(* Logix 5000 project; controller p65 vendor 1 type 14 code 85 rev 20.11; software revision 20.01; part 2 of 7 *)
(* tags used below, declared in another part *)
   BatterybattCurrent : ALIAS FOR REAL00_0;
   BatterybattCurrentHILS : ALIAS FOR plc1_local_3[4];
   Batterybattcurrentoffset : REAL;
   BatterybattCurrentRaw : ALIAS FOR Local:1:I.Ch4Data;
   BatterybattPower : ALIAS FOR REAL00_1;
   BatterybattVoltage : ALIAS FOR REAL00_2;
   BatterybattVoltageHILS : ALIAS FOR plc1_local_3[5];
   BatterybattVoltageRaw : ALIAS FOR Local:1:I.Ch0Data;
   BatterycanSupplyPower : ALIAS FOR DINT00_22.0;
   Batterycharge : ALIAS FOR REAL00_3;
   BatterychargeCurrent : ALIAS FOR REAL00_4;
   BatterychargeToGo : ALIAS FOR REAL00_5;
   BatterychargingTimer : ALIAS FOR CLTIMER00_0;
   BatterycomputeAddition : ALIAS FOR DINT00_22.7;
   BatterycomputeSubtraction : ALIAS FOR DINT00_22.8;
   BatterydecideToCharge : ALIAS FOR DINT00_22.15;
   BatterydecideToDisconnect : ALIAS FOR DINT00_22.16;
   BatterydeltaCharge : ALIAS FOR REAL00_6;
   BatterydischargeCurrent : ALIAS FOR REAL00_7;
   BatterydischargingTimer : ALIAS FOR CLTIMER00_1;
   BatterydisconnectedTimer : ALIAS FOR CLTIMER00_2;
   Batteryefficiency : ALIAS FOR REAL00_8;
   Batteryfraction : ALIAS FOR REAL00_9;
   BatteryfractionCharged : ALIAS FOR REAL00_10;
   BatteryfractionChargedEstimate : ALIAS FOR REAL00_11;
   BatteryfractionToGo : ALIAS FOR REAL00_12;
   BatteryfullCharge : ALIAS FOR REAL00_13;
   BatteryfullChargeCurrent : ALIAS FOR REAL00_14;
   BatterygeneralTimer : ALIAS FOR CLTIMER00_3;
   BatterygridCurrent : ALIAS FOR REAL00_15;
   BatterygridCurrentabs : REAL;
   BatterygridCurrentHILS : ALIAS FOR plc1_local_3[2];
   Batterygridcurrentoffset : REAL;
   BatterygridCurrentRaw : ALIAS FOR Local:1:I.Ch5Data;
   BatterygridPower : ALIAS FOR REAL00_16;
   BatterygridVoltage : ALIAS FOR REAL00_17;
   BatterygridVoltageHILS : ALIAS FOR plc1_local_3[3];
   BatterygridVoltageRaw : ALIAS FOR Local:1:I.Ch9Data;
   BatteryintReqCharge : ALIAS FOR DINT00_22.17;
   BatteryintReqDischarge : ALIAS FOR DINT00_22.18;
   BatteryintReqDisconnect : ALIAS FOR DINT00_22.19;
   BatteryisCharging : ALIAS FOR DINT00_22.20;
   BatteryisDischarging : ALIAS FOR DINT00_22.21;
   BatteryisDisconnected : ALIAS FOR DINT00_22.22;
   BatteryisFullyCharged : ALIAS FOR DINT00_22.23;
   BatteryisFunctional : ALIAS FOR DINT00_22.24;
   BatterylastChargingTime : ALIAS FOR DINT00_0;
   BatterylastDischargingTime : ALIAS FOR DINT00_1;
   BatterylastDisconnectedTime : ALIAS FOR DINT00_2;
   BatterylastFractionChargedDelta : ALIAS FOR REAL00_18;
   BatterylastIntReqCharge : ALIAS FOR DINT00_22.25;
   BatterylastIntReqDischarge : ALIAS FOR DINT00_22.26;
   BatterylastIntReqDisconnect : ALIAS FOR DINT00_22.27;
   BatterylowestSOC : ALIAS FOR REAL00_19;
   Batterymultiplier : ALIAS FOR REAL00_20;
   BatterynominalDischargeCurrent : ALIAS FOR REAL00_21;
   BatteryocVoltage : ALIAS FOR REAL00_22;
   BatteryoutOfOperationalRange : ALIAS FOR DINT00_22.28;
   BatterypeukertLessOne : ALIAS FOR REAL00_23;
   Batteryproduct : ALIAS FOR REAL00_24;
   BatteryreqCharge : ALIAS FOR DINT00_22.29;
   BatteryreqDischarge : ALIAS FOR DINT00_22.30;
   BatteryreqDisconnect : ALIAS FOR DINT00_22.31;
   BatteryreqInitialize : ALIAS FOR DINT00_23.0;
   BatterysettlingTimer : ALIAS FOR CLTIMER00_4;
   Batterysoc : ALIAS FOR REAL00_25;
   BatterysocToGo : ALIAS FOR REAL00_26;
   BatterySOCTooLowEventFail : ALIAS FOR DINT00_23.1;
   BatterySOCTooLowEventSuccess : ALIAS FOR DINT00_23.2;
   BatterySOCTooLowFailTimer : ALIAS FOR CLTIMER00_5;
   BatterySOCTooLowInProcess : ALIAS FOR DINT00_23.3;
   BatterySOCTooLowMsg : ALIAS FOR MESSAGE00_0;
   BatterySOCTooLowSuccessTimer : ALIAS FOR CLTIMER00_6;
   BatterytimeSinceLastMeasurement : ALIAS FOR REAL00_27;
   BatterytimeToLowestSOC : ALIAS FOR REAL00_28;
   BatteryunambiguousCommand : ALIAS FOR DINT00_23.4;
   CBclose : ALIAS FOR Local:3:O.Data.15;
   CBcloseHILS : ALIAS FOR plc1_local_6[0].14;
   CBcloseProxy : ALIAS FOR DINT00_22.1;
   CBintReqClose : ALIAS FOR DINT00_22.2;
   CBisClosed : ALIAS FOR DINT00_22.3;
   CBisOpen : ALIAS FOR DINT00_22.4;
   CBreqClose : ALIAS FOR DINT00_22.5;
   CBreqOpen : ALIAS FOR DINT00_22.6;
   Commaccum : ALIAS FOR REAL00_31;
   CommBattempt : ALIAS FOR DINT00_3;
   CommBclose : ALIAS FOR Local:3:O.Data.11;
   CommBcloseHILS : ALIAS FOR plc1_local_6[0].11;
   CommBcloseProxy : ALIAS FOR DINT00_23.12;
   CommBdeadBand : ALIAS FOR REAL00_32;
   CommBfailedToOpen : ALIAS FOR DINT00_23.13;
   CommBintForceOpen : ALIAS FOR DINT00_23.14;
   CommBintReqClose : ALIAS FOR DINT00_23.15;
   CommBisClosed : ALIAS FOR DINT00_23.16;
   CommBisOpen : ALIAS FOR DINT00_23.17;
   CommBmaxAttempts : ALIAS FOR DINT00_4;
   CommBmaxLoadCurrent : ALIAS FOR REAL00_33;
   CommBopenTimer : ALIAS FOR CLTIMER00_7;
   CommBreqClose : ALIAS FOR DINT00_23.18;
   CommBreqOpen : ALIAS FOR DINT00_23.19;
   CommBreqReset : ALIAS FOR DINT00_23.20;
   CommBretriesFailed : ALIAS FOR DINT00_23.21;
   CommBtooMuchCurrent : ALIAS FOR DINT00_23.22;
   CommBunexpectedLowCurrent : ALIAS FOR DINT00_23.23;
   CommcanNotifyUser : ALIAS FOR DINT00_23.24;
   CommcommandChanged : ALIAS FOR DINT00_23.25;
   CommcommandChangedTimer : ALIAS FOR CLTIMER00_8;
   Commcurrent : ALIAS FOR REAL00_34;
   CommcurrentHILS : ALIAS FOR plc1_local_3[8];
   CommcurrentRaw : ALIAS FOR Local:1:I.Ch10Data;
   Commdeadband : ALIAS FOR REAL00_35;
   Commdifference : ALIAS FOR REAL00_36;
   CommfailedToConnect : ALIAS FOR DINT00_23.26;
   CommfailedToDisconnect : ALIAS FOR DINT00_23.27;
   CommintReqConnect : ALIAS FOR DINT00_23.28;
   CommisConnected : ALIAS FOR DINT00_23.29;
   CommisDisconnected : ALIAS FOR DINT00_23.30;
   CommnotificationTimer : ALIAS FOR CLTIMER00_44;
   CommOverCurrentConditionEventFail : ALIAS FOR DINT00_27.13;
   CommOverCurrentConditionEventSuccess : ALIAS FOR DINT00_27.14;
   CommOverCurrentConditionFailTimer : ALIAS FOR CLTIMER00_45;
   CommOverCurrentConditionInProcess : ALIAS FOR DINT00_27.15;
   CommOverCurrentConditionMsg : ALIAS FOR MESSAGE00_11;
   CommOverCurrentConditionSuccessTimer : ALIAS FOR CLTIMER00_46;
   Commpower : ALIAS FOR REAL00_102;
   CommreqConnect : ALIAS FOR DINT00_27.16;
   CommreqDisconnect : ALIAS FOR DINT00_27.17;
   CommsampleNow : ALIAS FOR DINT00_27.18;
   CommsampleTimer : ALIAS FOR CLTIMER00_47;
   Commtotal : ALIAS FOR REAL00_103;
   CommtotalTooLarge : ALIAS FOR DINT00_27.19;
   CommtotalTooSmall : ALIAS FOR DINT00_27.20;
   CommuserNotified : ALIAS FOR DINT00_27.21;
   Commvoltage : ALIAS FOR REAL00_104;
   CommvoltageHILS : ALIAS FOR plc1_local_3[9];
   CommvoltageRaw : ALIAS FOR Local:2:I.Ch7Data;
   DBclose : ALIAS FOR Local:3:O.Data.14;
   DBcloseHILS : ALIAS FOR plc1_local_6[0].13;
   DBcloseProxy : ALIAS FOR DINT00_22.9;
   DBintReqClose : ALIAS FOR DINT00_22.10;
   DBisClosed : ALIAS FOR DINT00_22.11;
   DBisOpen : ALIAS FOR DINT00_22.12;
   DBreqClose : ALIAS FOR DINT00_22.13;
   DBreqOpen : ALIAS FOR DINT00_22.14;
   DCMicroGridisSimulating : ALIAS FOR DINT00_23.10;
   DCMicroGridsourcesProvidingExcessPower : ALIAS FOR DINT00_33.7;
   Load01current : ALIAS FOR REAL00_39;
   Load02current : ALIAS FOR REAL00_52;
   Load03current : ALIAS FOR REAL00_65;
   Load04current : ALIAS FOR REAL00_78;
   Load05current : ALIAS FOR REAL00_91;
   LoadslowVoltage : ALIAS FOR DINT00_27.23;
   UsingAgents : BOOL;

PROGRAM Battery   (* main routine Battery *)

ROUTINE Battery   (* ladder *)
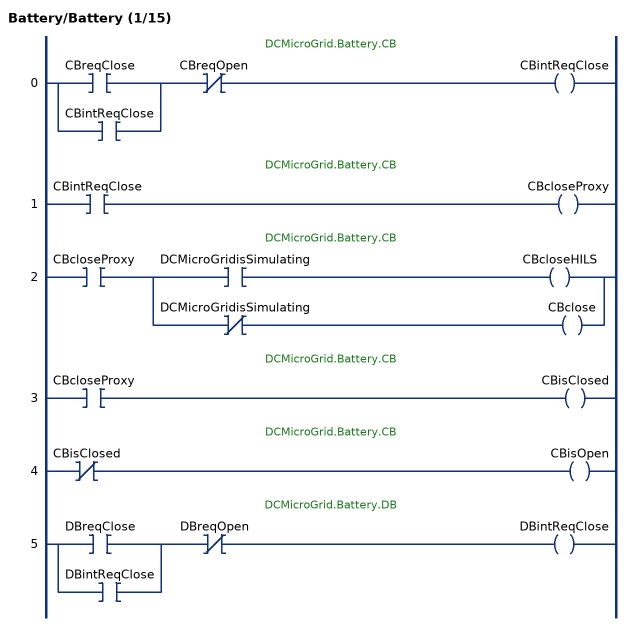
   // DCMicroGrid.Battery.CB
   0: [XIC(CBreqClose) ,XIC(CBintReqClose) ]XIO(CBreqOpen)OTE(CBintReqClose);
   // DCMicroGrid.Battery.CB
   1: XIC(CBintReqClose)OTE(CBcloseProxy);
   // DCMicroGrid.Battery.CB
   2: XIC(CBcloseProxy)[XIC(DCMicroGridisSimulating) OTE(CBcloseHILS) ,XIO(DCMicroGridisSimulating) OTE(CBclose) ];
   // DCMicroGrid.Battery.CB
   3: XIC(CBcloseProxy)OTE(CBisClosed);
   // DCMicroGrid.Battery.CB
   4: XIO(CBisClosed)OTE(CBisOpen);
   // DCMicroGrid.Battery.DB
   5: [XIC(DBreqClose) ,XIC(DBintReqClose) ]XIO(DBreqOpen)OTE(DBintReqClose);
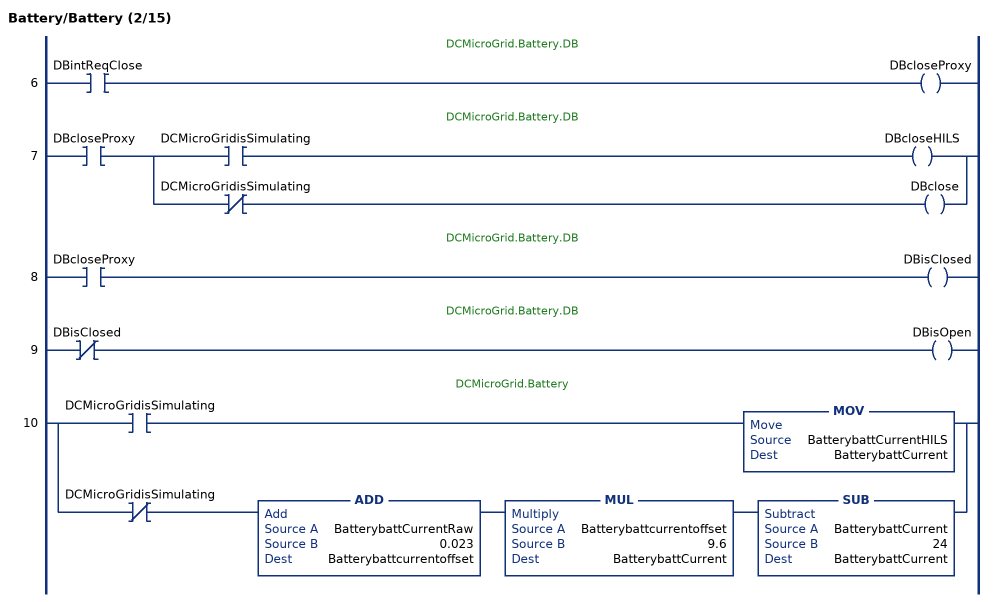
   // DCMicroGrid.Battery.DB
   6: XIC(DBintReqClose)OTE(DBcloseProxy);
   // DCMicroGrid.Battery.DB
   7: XIC(DBcloseProxy)[XIC(DCMicroGridisSimulating) OTE(DBcloseHILS) ,XIO(DCMicroGridisSimulating) OTE(DBclose) ];
   // DCMicroGrid.Battery.DB
   8: XIC(DBcloseProxy)OTE(DBisClosed);
   // DCMicroGrid.Battery.DB
   9: XIO(DBisClosed)OTE(DBisOpen);
   // DCMicroGrid.Battery
   10: [XIC(DCMicroGridisSimulating) MOV(BatterybattCurrentHILS,BatterybattCurrent) ,XIO(DCMicroGridisSimulating) ADD(BatterybattCurrentRaw,0.023,Batterybattcurrentoffset) MUL(Batterybattcurrentoffset,9.6,BatterybattCurrent) SUB(BatterybattCurrent,24,BatterybattCurrent) ];
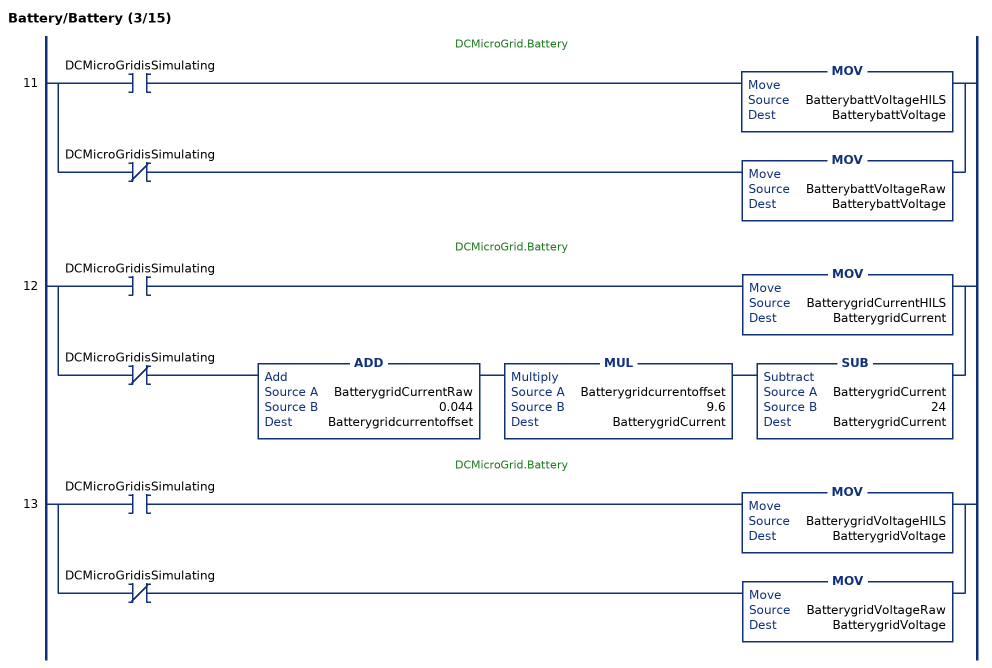
   // DCMicroGrid.Battery
   11: [XIC(DCMicroGridisSimulating) MOV(BatterybattVoltageHILS,BatterybattVoltage) ,XIO(DCMicroGridisSimulating) MOV(BatterybattVoltageRaw,BatterybattVoltage) ];
   // DCMicroGrid.Battery
   12: [XIC(DCMicroGridisSimulating) MOV(BatterygridCurrentHILS,BatterygridCurrent) ,XIO(DCMicroGridisSimulating) ADD(BatterygridCurrentRaw,0.044,Batterygridcurrentoffset) MUL(Batterygridcurrentoffset,9.6,BatterygridCurrent) SUB(BatterygridCurrent,24,BatterygridCurrent) ];
   // DCMicroGrid.Battery
   13: [XIC(DCMicroGridisSimulating) MOV(BatterygridVoltageHILS,BatterygridVoltage) ,XIO(DCMicroGridisSimulating) MOV(BatterygridVoltageRaw,BatterygridVoltage) ];
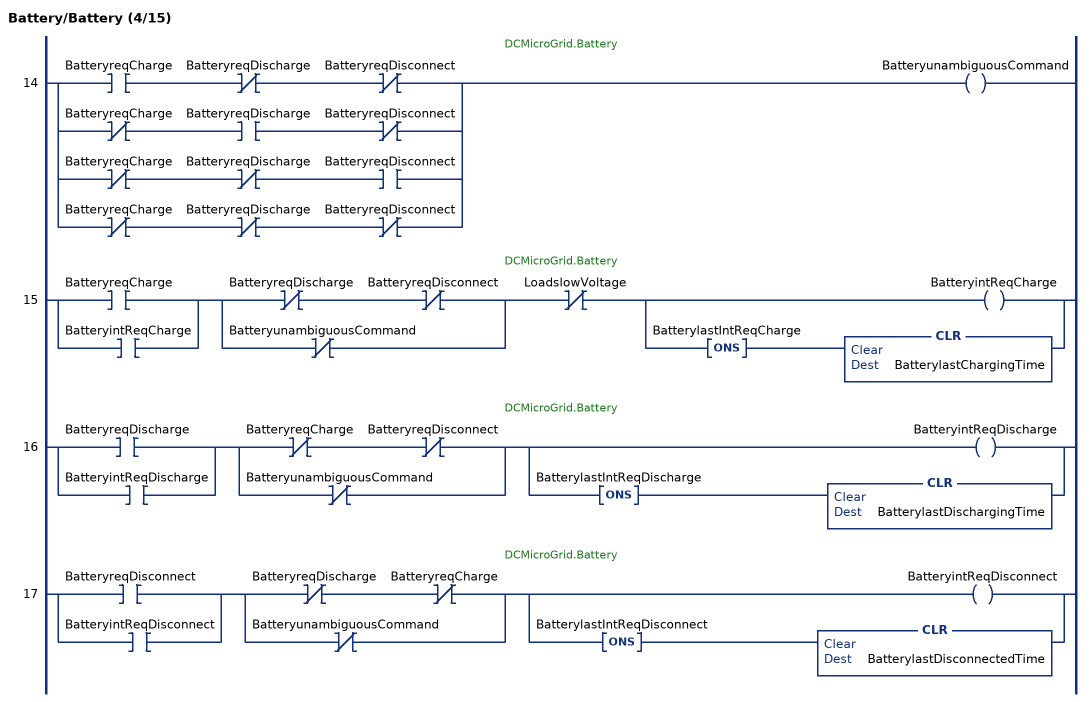
   // DCMicroGrid.Battery
   14: [XIC(BatteryreqCharge) XIO(BatteryreqDischarge) XIO(BatteryreqDisconnect) ,XIO(BatteryreqCharge) XIC(BatteryreqDischarge) XIO(BatteryreqDisconnect) ,XIO(BatteryreqCharge) XIO(BatteryreqDischarge) XIC(BatteryreqDisconnect) ,XIO(BatteryreqCharge) XIO(BatteryreqDischarge) XIO(BatteryreqDisconnect) ]OTE(BatteryunambiguousCommand);
   // DCMicroGrid.Battery
   15: [XIC(BatteryreqCharge) ,XIC(BatteryintReqCharge) ][XIO(BatteryreqDischarge) XIO(BatteryreqDisconnect) ,XIO(BatteryunambiguousCommand) ]XIO(LoadslowVoltage)[OTE(BatteryintReqCharge) ,ONS(BatterylastIntReqCharge) CLR(BatterylastChargingTime) ];
   // DCMicroGrid.Battery
   16: [XIC(BatteryreqDischarge) ,XIC(BatteryintReqDischarge) ][XIO(BatteryreqCharge) XIO(BatteryreqDisconnect) ,XIO(BatteryunambiguousCommand) ][OTE(BatteryintReqDischarge) ,ONS(BatterylastIntReqDischarge) CLR(BatterylastDischargingTime) ];
   // DCMicroGrid.Battery
   17: [XIC(BatteryreqDisconnect) ,XIC(BatteryintReqDisconnect) ][XIO(BatteryreqDischarge) XIO(BatteryreqCharge) ,XIO(BatteryunambiguousCommand) ][OTE(BatteryintReqDisconnect) ,ONS(BatterylastIntReqDisconnect) CLR(BatterylastDisconnectedTime) ];
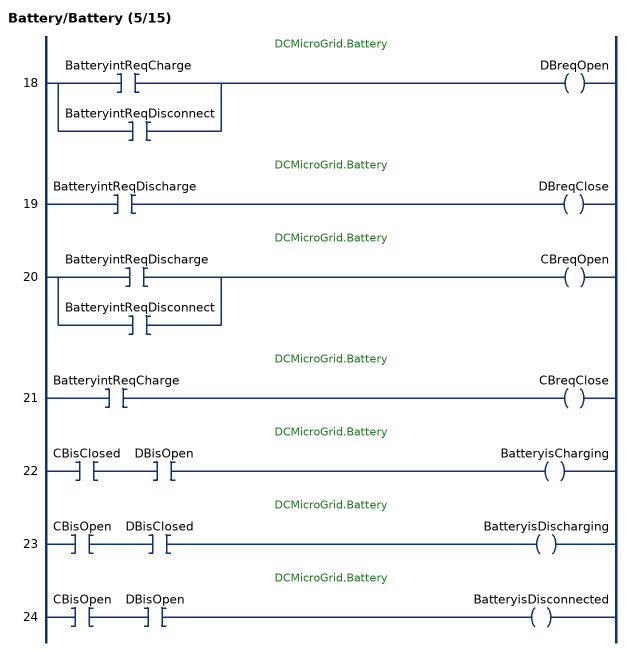
   // DCMicroGrid.Battery
   18: [XIC(BatteryintReqCharge) ,XIC(BatteryintReqDisconnect) ]OTE(DBreqOpen);
   // DCMicroGrid.Battery
   19: XIC(BatteryintReqDischarge)OTE(DBreqClose);
   // DCMicroGrid.Battery
   20: [XIC(BatteryintReqDischarge) ,XIC(BatteryintReqDisconnect) ]OTE(CBreqOpen);
   // DCMicroGrid.Battery
   21: XIC(BatteryintReqCharge)OTE(CBreqClose);
   // DCMicroGrid.Battery
   22: XIC(CBisClosed)XIC(DBisOpen)OTE(BatteryisCharging);
   // DCMicroGrid.Battery
   23: XIC(CBisOpen)XIC(DBisClosed)OTE(BatteryisDischarging);
   // DCMicroGrid.Battery
   24: XIC(CBisOpen)XIC(DBisOpen)OTE(BatteryisDisconnected);
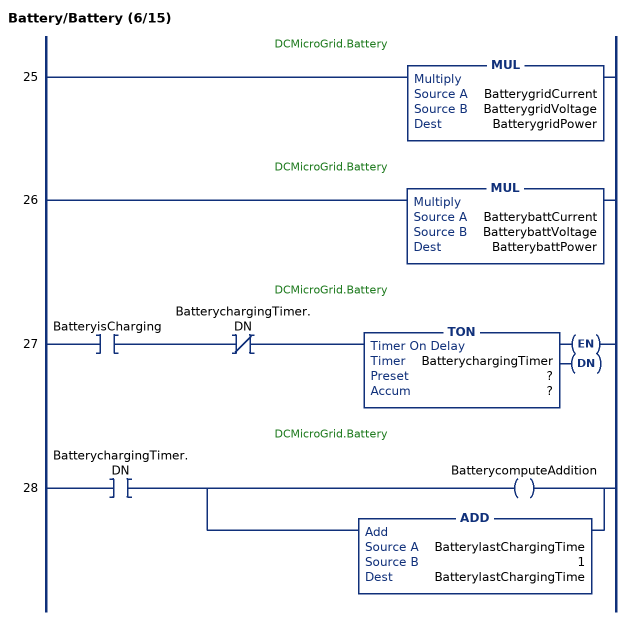
   // DCMicroGrid.Battery
   25: MUL(BatterygridCurrent,BatterygridVoltage,BatterygridPower);
   // DCMicroGrid.Battery
   26: MUL(BatterybattCurrent,BatterybattVoltage,BatterybattPower);
   // DCMicroGrid.Battery
   27: XIC(BatteryisCharging)XIO(BatterychargingTimer.DN)TON(BatterychargingTimer,?,?);
   // DCMicroGrid.Battery
   28: XIC(BatterychargingTimer.DN)[OTE(BatterycomputeAddition) ,ADD(BatterylastChargingTime,1,BatterylastChargingTime) ];
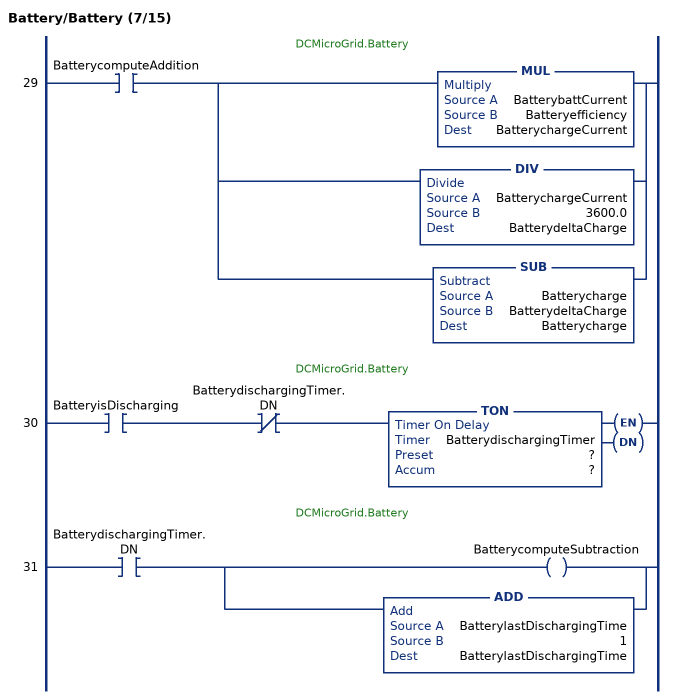
   // DCMicroGrid.Battery
   29: XIC(BatterycomputeAddition)[MUL(BatterybattCurrent,Batteryefficiency,BatterychargeCurrent) ,DIV(BatterychargeCurrent,3600.0,BatterydeltaCharge) ,SUB(Batterycharge,BatterydeltaCharge,Batterycharge) ];
   // DCMicroGrid.Battery
   30: XIC(BatteryisDischarging)XIO(BatterydischargingTimer.DN)TON(BatterydischargingTimer,?,?);
   // DCMicroGrid.Battery
   31: XIC(BatterydischargingTimer.DN)[OTE(BatterycomputeSubtraction) ,ADD(BatterylastDischargingTime,1,BatterylastDischargingTime) ];
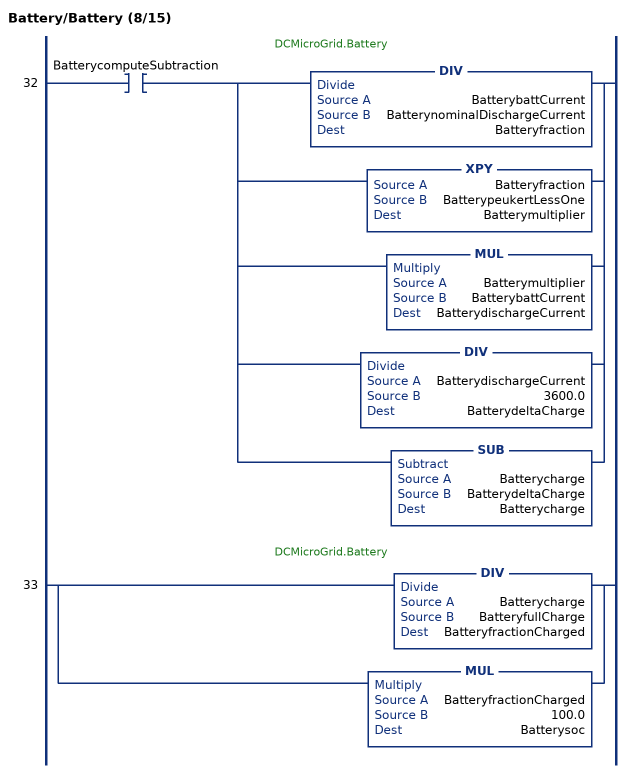
   // DCMicroGrid.Battery
   32: XIC(BatterycomputeSubtraction)[DIV(BatterybattCurrent,BatterynominalDischargeCurrent,Batteryfraction) ,XPY(Batteryfraction,BatterypeukertLessOne,Batterymultiplier) ,MUL(Batterymultiplier,BatterybattCurrent,BatterydischargeCurrent) ,DIV(BatterydischargeCurrent,3600.0,BatterydeltaCharge) ,SUB(Batterycharge,BatterydeltaCharge,Batterycharge) ];
   // DCMicroGrid.Battery
   33: [DIV(Batterycharge,BatteryfullCharge,BatteryfractionCharged) ,MUL(BatteryfractionCharged,100.0,Batterysoc) ];
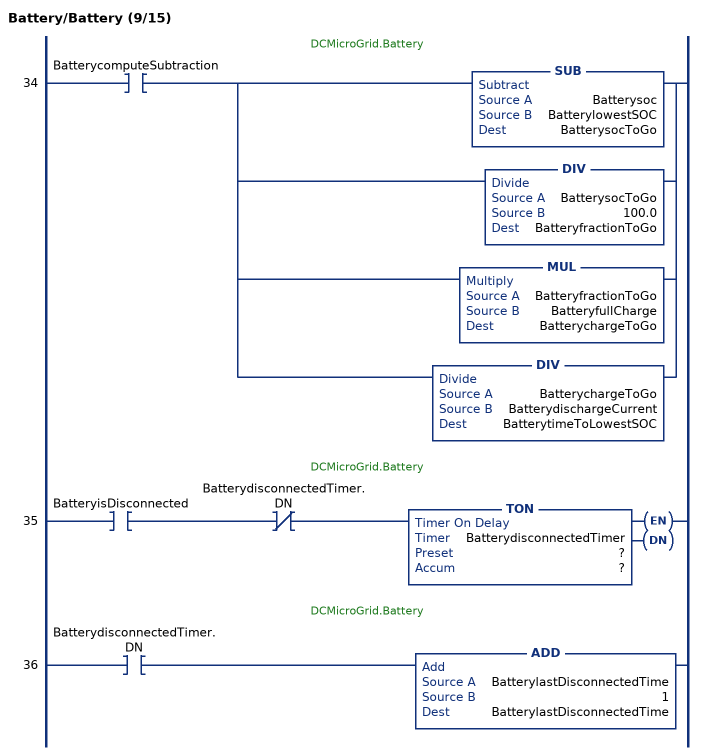
   // DCMicroGrid.Battery
   34: XIC(BatterycomputeSubtraction)[SUB(Batterysoc,BatterylowestSOC,BatterysocToGo) ,DIV(BatterysocToGo,100.0,BatteryfractionToGo) ,MUL(BatteryfractionToGo,BatteryfullCharge,BatterychargeToGo) ,DIV(BatterychargeToGo,BatterydischargeCurrent,BatterytimeToLowestSOC) ];
   // DCMicroGrid.Battery
   35: XIC(BatteryisDisconnected)XIO(BatterydisconnectedTimer.DN)TON(BatterydisconnectedTimer,?,?);
   // DCMicroGrid.Battery
   36: XIC(BatterydisconnectedTimer.DN)ADD(BatterylastDisconnectedTime,1,BatterylastDisconnectedTime);
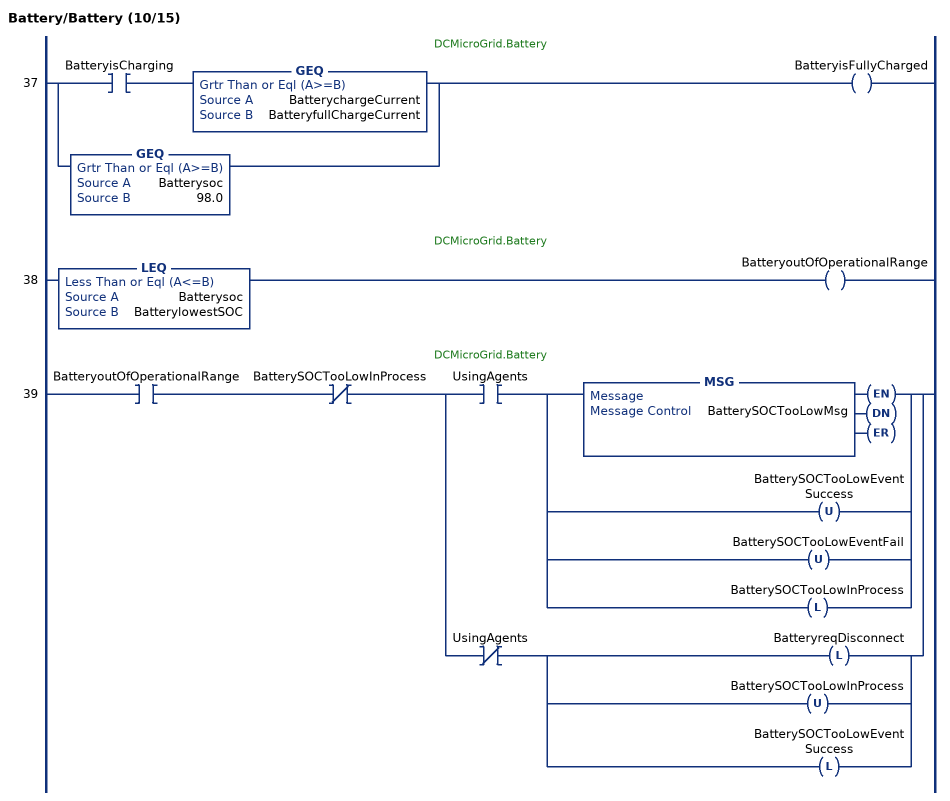
   // DCMicroGrid.Battery
   37: [XIC(BatteryisCharging) GEQ(BatterychargeCurrent,BatteryfullChargeCurrent) ,GEQ(Batterysoc,98.0) ]OTE(BatteryisFullyCharged);
   // DCMicroGrid.Battery
   38: LEQ(Batterysoc,BatterylowestSOC)OTE(BatteryoutOfOperationalRange);
   // DCMicroGrid.Battery
   39: XIC(BatteryoutOfOperationalRange)XIO(BatterySOCTooLowInProcess)[XIC(UsingAgents) [MSG(BatterySOCTooLowMsg) ,OTU(BatterySOCTooLowEventSuccess) ,OTU(BatterySOCTooLowEventFail) ,OTL(BatterySOCTooLowInProcess) ] ,XIO(UsingAgents) [OTL(BatteryreqDisconnect) ,OTU(BatterySOCTooLowInProcess) ,OTL(BatterySOCTooLowEventSuccess) ] ];
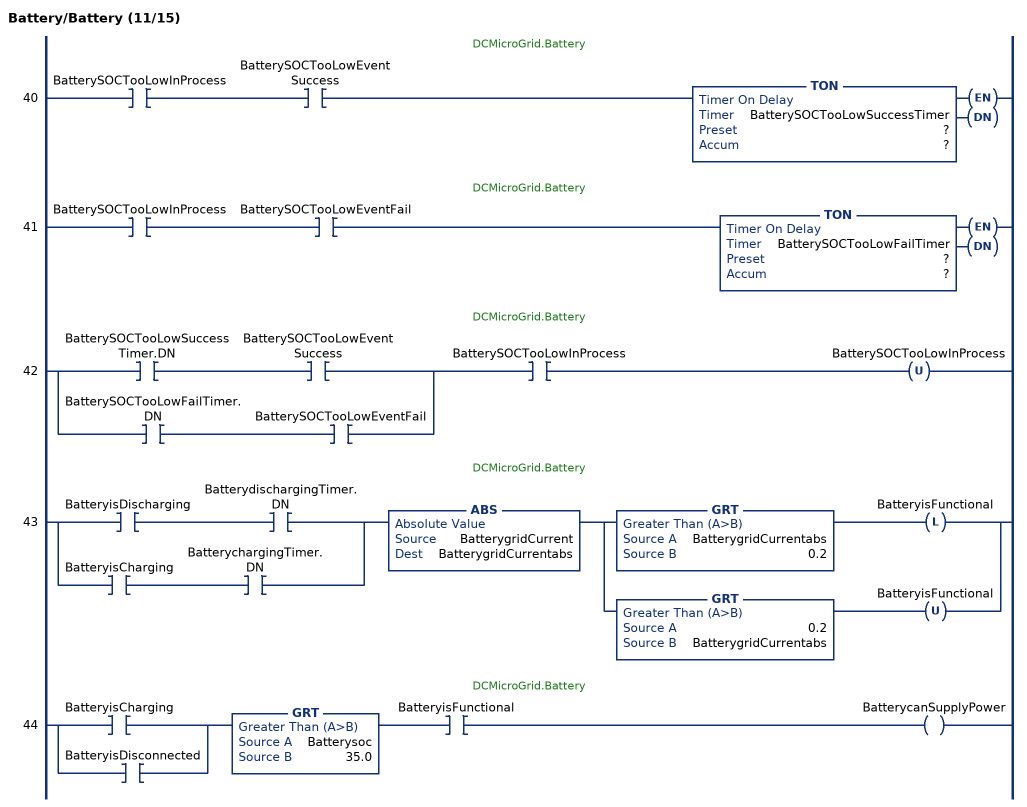
   // DCMicroGrid.Battery
   40: XIC(BatterySOCTooLowInProcess)XIC(BatterySOCTooLowEventSuccess)TON(BatterySOCTooLowSuccessTimer,?,?);
   // DCMicroGrid.Battery
   41: XIC(BatterySOCTooLowInProcess)XIC(BatterySOCTooLowEventFail)TON(BatterySOCTooLowFailTimer,?,?);
   // DCMicroGrid.Battery
   42: [XIC(BatterySOCTooLowSuccessTimer.DN) XIC(BatterySOCTooLowEventSuccess) ,XIC(BatterySOCTooLowFailTimer.DN) XIC(BatterySOCTooLowEventFail) ]XIC(BatterySOCTooLowInProcess)OTU(BatterySOCTooLowInProcess);
   // DCMicroGrid.Battery
   43: [XIC(BatteryisDischarging) XIC(BatterydischargingTimer.DN) ,XIC(BatteryisCharging) XIC(BatterychargingTimer.DN) ]ABS(BatterygridCurrent,BatterygridCurrentabs)[GRT(BatterygridCurrentabs,0.2) OTL(BatteryisFunctional) ,GRT(0.2,BatterygridCurrentabs) OTU(BatteryisFunctional) ];
   // DCMicroGrid.Battery
   44: [XIC(BatteryisCharging) ,XIC(BatteryisDisconnected) ]GRT(Batterysoc,35.0)XIC(BatteryisFunctional)OTE(BatterycanSupplyPower);
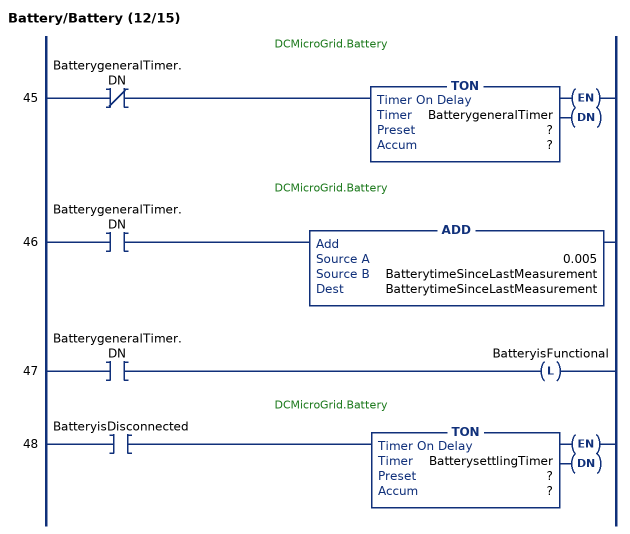
   // DCMicroGrid.Battery
   45: XIO(BatterygeneralTimer.DN)TON(BatterygeneralTimer,?,?);
   // DCMicroGrid.Battery
   46: XIC(BatterygeneralTimer.DN)ADD(0.005,BatterytimeSinceLastMeasurement,BatterytimeSinceLastMeasurement);
   47: XIC(BatterygeneralTimer.DN)OTL(BatteryisFunctional);
   // DCMicroGrid.Battery
   48: XIC(BatteryisDisconnected)TON(BatterysettlingTimer,?,?);
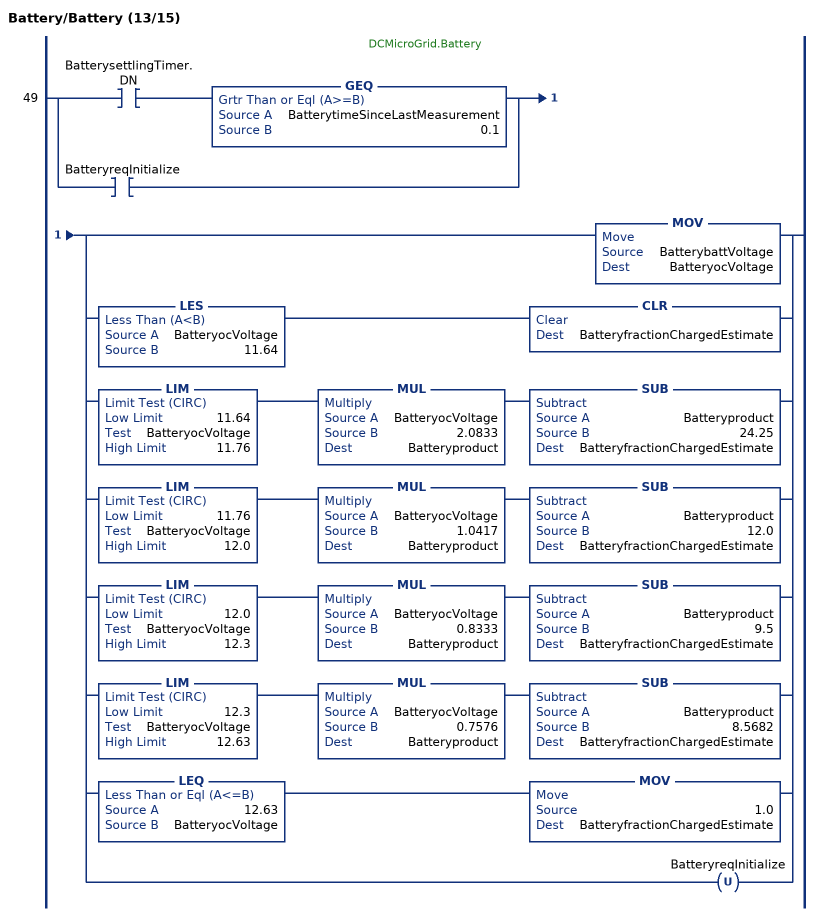
   // DCMicroGrid.Battery
   49: [XIC(BatterysettlingTimer.DN) GEQ(BatterytimeSinceLastMeasurement,0.1) ,XIC(BatteryreqInitialize) ][MOV(BatterybattVoltage,BatteryocVoltage) ,LES(BatteryocVoltage,11.64) CLR(BatteryfractionChargedEstimate) ,LIM(11.64,BatteryocVoltage,11.76) MUL(BatteryocVoltage,2.0833,Batteryproduct) SUB(Batteryproduct,24.25,BatteryfractionChargedEstimate) ,LIM(11.76,BatteryocVoltage,12.0) MUL(BatteryocVoltage,1.0417,Batteryproduct) SUB(Batteryproduct,12.0,BatteryfractionChargedEstimate) ,LIM(12.0,BatteryocVoltage,12.3) MUL(BatteryocVoltage,0.8333,Batteryproduct) SUB(Batteryproduct,9.5,BatteryfractionChargedEstimate) ,LIM(12.3,BatteryocVoltage,12.63) MUL(BatteryocVoltage,0.7576,Batteryproduct) SUB(Batteryproduct,8.5682,BatteryfractionChargedEstimate) ,LEQ(12.63,BatteryocVoltage) MOV(1.0,BatteryfractionChargedEstimate) ,OTU(BatteryreqInitialize) ];
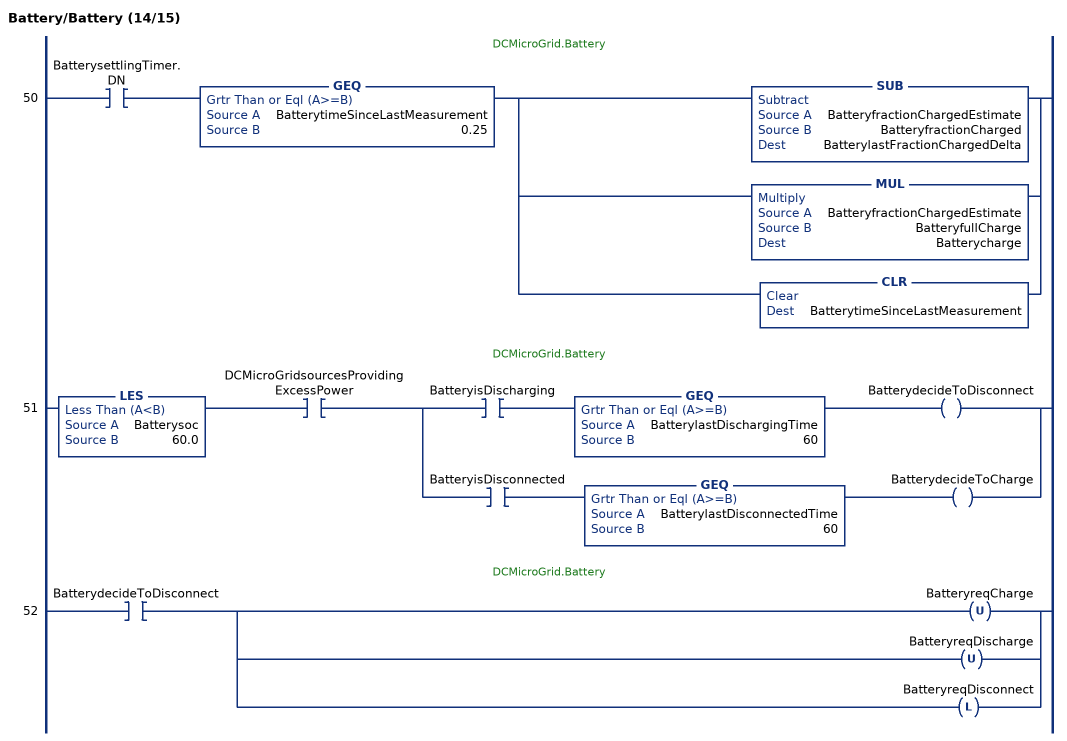
   // DCMicroGrid.Battery
   50: XIC(BatterysettlingTimer.DN)GEQ(BatterytimeSinceLastMeasurement,0.25)[SUB(BatteryfractionChargedEstimate,BatteryfractionCharged,BatterylastFractionChargedDelta) ,MUL(BatteryfractionChargedEstimate,BatteryfullCharge,Batterycharge) ,CLR(BatterytimeSinceLastMeasurement) ];
   // DCMicroGrid.Battery
   51: LES(Batterysoc,60.0)XIC(DCMicroGridsourcesProvidingExcessPower)[XIC(BatteryisDischarging) GEQ(BatterylastDischargingTime,60) OTE(BatterydecideToDisconnect) ,XIC(BatteryisDisconnected) GEQ(BatterylastDisconnectedTime,60) OTE(BatterydecideToCharge) ];
   // DCMicroGrid.Battery
   52: XIC(BatterydecideToDisconnect)[OTU(BatteryreqCharge) ,OTU(BatteryreqDischarge) ,OTL(BatteryreqDisconnect) ];
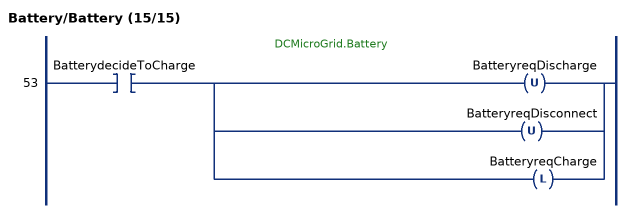
   // DCMicroGrid.Battery
   53: XIC(BatterydecideToCharge)[OTU(BatteryreqDischarge) ,OTU(BatteryreqDisconnect) ,OTL(BatteryreqCharge) ];
END_ROUTINE
END_PROGRAM

PROGRAM Comm   (* main routine Comm *)

ROUTINE Comm   (* ladder *)
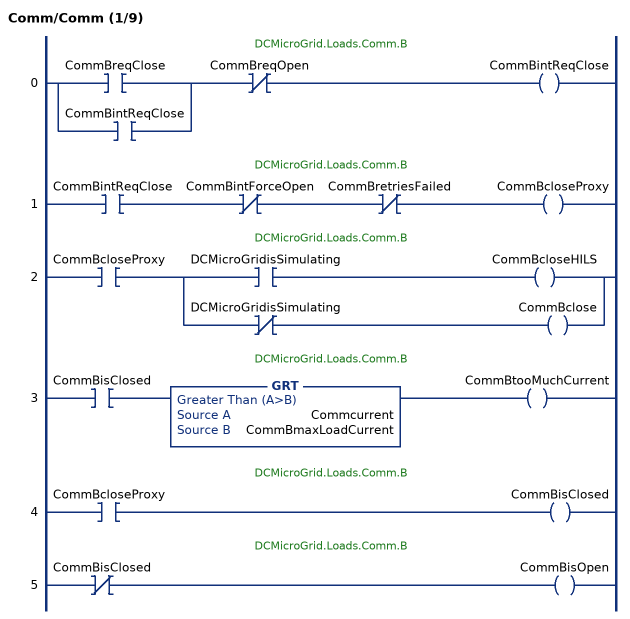
   // DCMicroGrid.Loads.Comm.B
   0: [XIC(CommBreqClose) ,XIC(CommBintReqClose) ]XIO(CommBreqOpen)OTE(CommBintReqClose);
   // DCMicroGrid.Loads.Comm.B
   1: XIC(CommBintReqClose)XIO(CommBintForceOpen)XIO(CommBretriesFailed)OTE(CommBcloseProxy);
   // DCMicroGrid.Loads.Comm.B
   2: XIC(CommBcloseProxy)[XIC(DCMicroGridisSimulating) OTE(CommBcloseHILS) ,XIO(DCMicroGridisSimulating) OTE(CommBclose) ];
   // DCMicroGrid.Loads.Comm.B
   3: XIC(CommBisClosed)GRT(Commcurrent,CommBmaxLoadCurrent)OTE(CommBtooMuchCurrent);
   // DCMicroGrid.Loads.Comm.B
   4: XIC(CommBcloseProxy)OTE(CommBisClosed);
   // DCMicroGrid.Loads.Comm.B
   5: XIO(CommBisClosed)OTE(CommBisOpen);
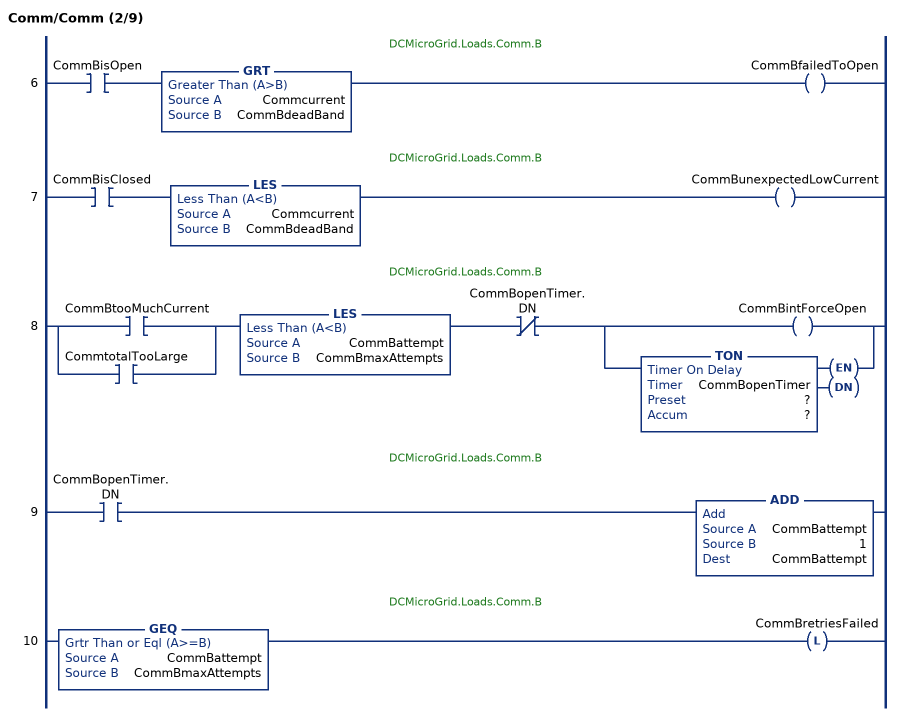
   // DCMicroGrid.Loads.Comm.B
   6: XIC(CommBisOpen)GRT(Commcurrent,CommBdeadBand)OTE(CommBfailedToOpen);
   // DCMicroGrid.Loads.Comm.B
   7: XIC(CommBisClosed)LES(Commcurrent,CommBdeadBand)OTE(CommBunexpectedLowCurrent);
   // DCMicroGrid.Loads.Comm.B
   8: [XIC(CommBtooMuchCurrent) ,XIC(CommtotalTooLarge) ]LES(CommBattempt,CommBmaxAttempts)XIO(CommBopenTimer.DN)[OTE(CommBintForceOpen) ,TON(CommBopenTimer,?,?) ];
   // DCMicroGrid.Loads.Comm.B
   9: XIC(CommBopenTimer.DN)ADD(CommBattempt,1,CommBattempt);
   // DCMicroGrid.Loads.Comm.B
   10: GEQ(CommBattempt,CommBmaxAttempts)OTL(CommBretriesFailed);
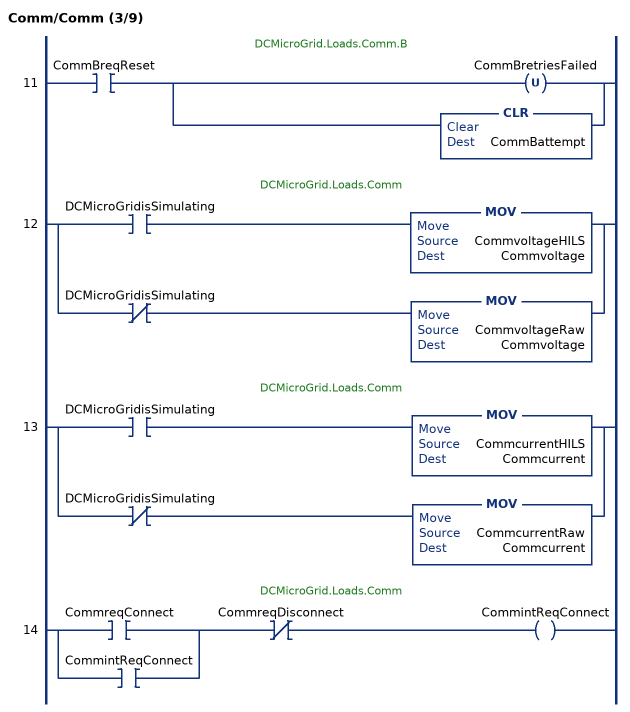
   // DCMicroGrid.Loads.Comm.B
   11: XIC(CommBreqReset)[OTU(CommBretriesFailed) ,CLR(CommBattempt) ];
   // DCMicroGrid.Loads.Comm
   12: [XIC(DCMicroGridisSimulating) MOV(CommvoltageHILS,Commvoltage) ,XIO(DCMicroGridisSimulating) MOV(CommvoltageRaw,Commvoltage) ];
   // DCMicroGrid.Loads.Comm
   13: [XIC(DCMicroGridisSimulating) MOV(CommcurrentHILS,Commcurrent) ,XIO(DCMicroGridisSimulating) MOV(CommcurrentRaw,Commcurrent) ];
   // DCMicroGrid.Loads.Comm
   14: [XIC(CommreqConnect) ,XIC(CommintReqConnect) ]XIO(CommreqDisconnect)OTE(CommintReqConnect);
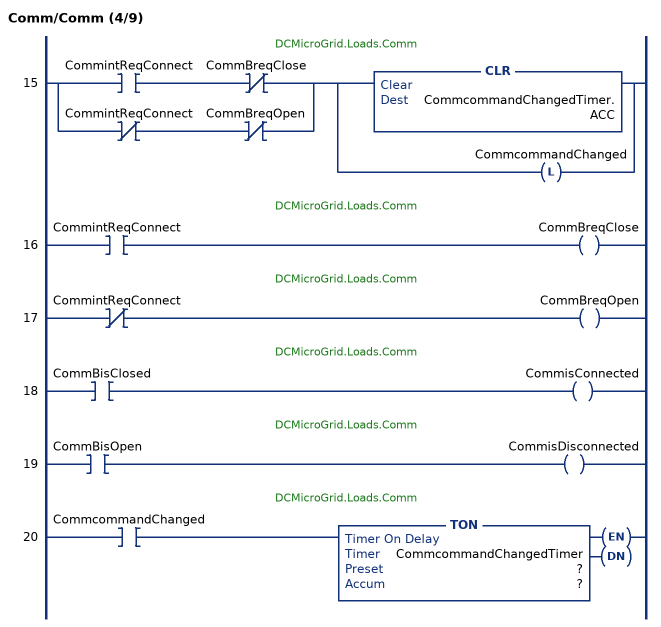
   // DCMicroGrid.Loads.Comm
   15: [XIC(CommintReqConnect) XIO(CommBreqClose) ,XIO(CommintReqConnect) XIO(CommBreqOpen) ][CLR(CommcommandChangedTimer.ACC) ,OTL(CommcommandChanged) ];
   // DCMicroGrid.Loads.Comm
   16: XIC(CommintReqConnect)OTE(CommBreqClose);
   // DCMicroGrid.Loads.Comm
   17: XIO(CommintReqConnect)OTE(CommBreqOpen);
   // DCMicroGrid.Loads.Comm
   18: XIC(CommBisClosed)OTE(CommisConnected);
   // DCMicroGrid.Loads.Comm
   19: XIC(CommBisOpen)OTE(CommisDisconnected);
   // DCMicroGrid.Loads.Comm
   20: XIC(CommcommandChanged)TON(CommcommandChangedTimer,?,?);
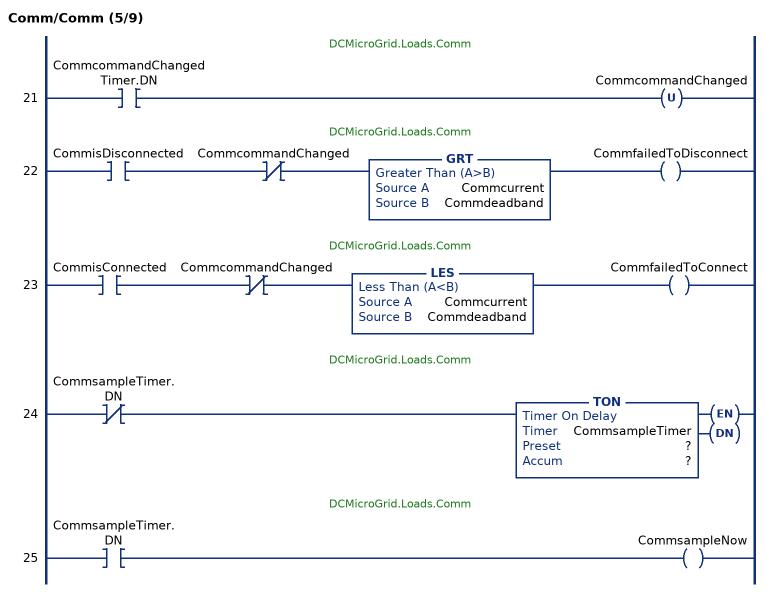
   // DCMicroGrid.Loads.Comm
   21: XIC(CommcommandChangedTimer.DN)OTU(CommcommandChanged);
   // DCMicroGrid.Loads.Comm
   22: XIC(CommisDisconnected)XIO(CommcommandChanged)GRT(Commcurrent,Commdeadband)OTE(CommfailedToDisconnect);
   // DCMicroGrid.Loads.Comm
   23: XIC(CommisConnected)XIO(CommcommandChanged)LES(Commcurrent,Commdeadband)OTE(CommfailedToConnect);
   // DCMicroGrid.Loads.Comm
   24: XIO(CommsampleTimer.DN)TON(CommsampleTimer,?,?);
   // DCMicroGrid.Loads.Comm
   25: XIC(CommsampleTimer.DN)OTE(CommsampleNow);
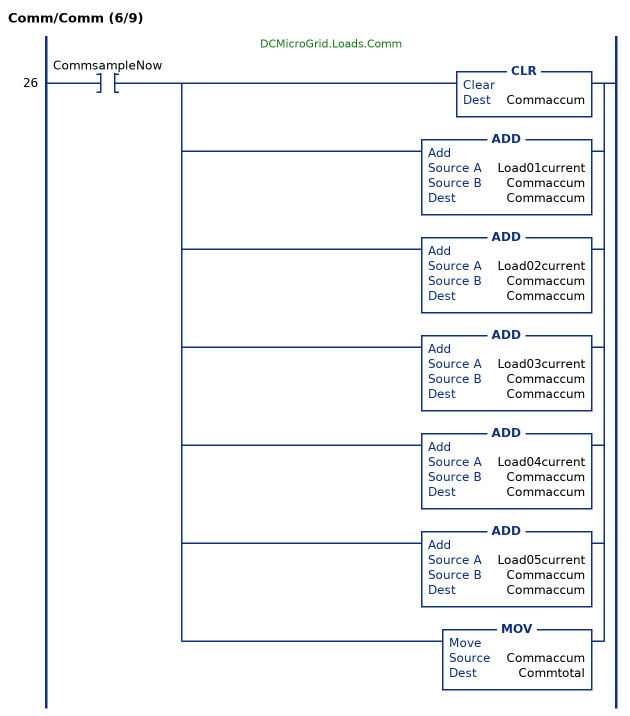
   // DCMicroGrid.Loads.Comm
   26: XIC(CommsampleNow)[CLR(Commaccum) ,[ADD(Load01current,Commaccum,Commaccum) ,ADD(Load02current,Commaccum,Commaccum) ,ADD(Load03current,Commaccum,Commaccum) ,ADD(Load04current,Commaccum,Commaccum) ,ADD(Load05current,Commaccum,Commaccum) ] ,MOV(Commaccum,Commtotal) ];
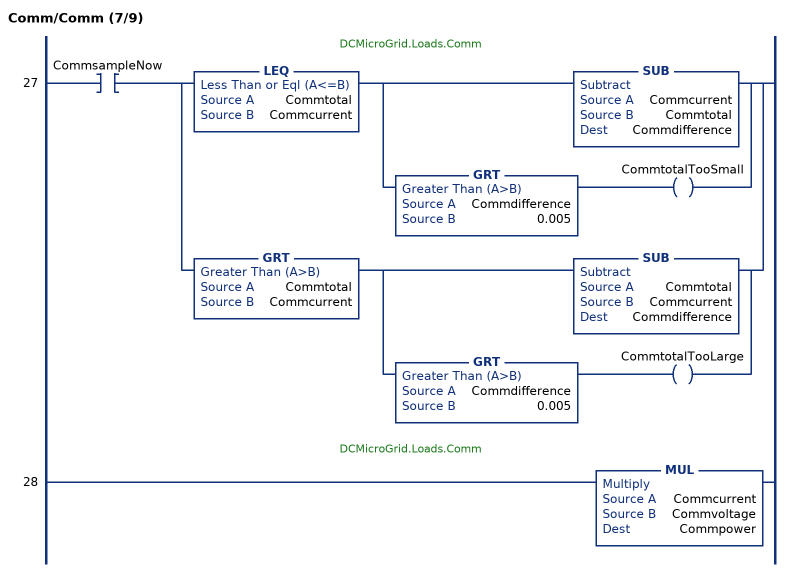
   // DCMicroGrid.Loads.Comm
   27: XIC(CommsampleNow)[LEQ(Commtotal,Commcurrent) [SUB(Commcurrent,Commtotal,Commdifference) ,GRT(Commdifference,0.005) OTE(CommtotalTooSmall) ] ,GRT(Commtotal,Commcurrent) [SUB(Commtotal,Commcurrent,Commdifference) ,GRT(Commdifference,0.005) OTE(CommtotalTooLarge) ] ];
   // DCMicroGrid.Loads.Comm
   28: MUL(Commcurrent,Commvoltage,Commpower);
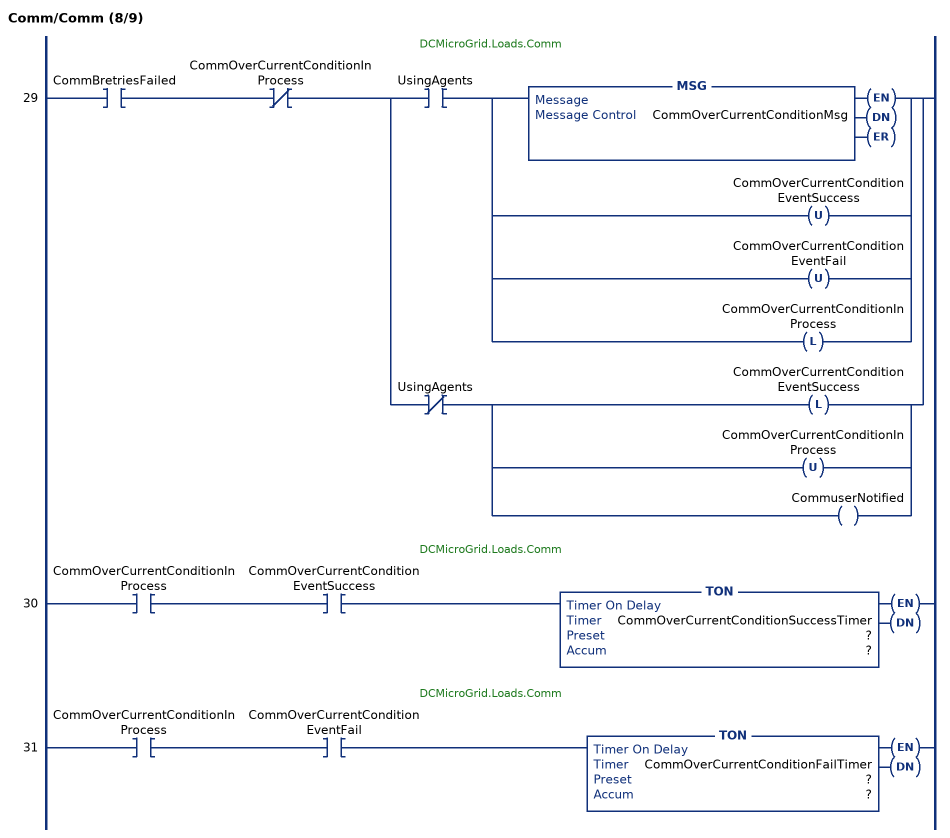
   // DCMicroGrid.Loads.Comm
   29: XIC(CommBretriesFailed)XIO(CommOverCurrentConditionInProcess)[XIC(UsingAgents) [MSG(CommOverCurrentConditionMsg) ,OTU(CommOverCurrentConditionEventSuccess) ,OTU(CommOverCurrentConditionEventFail) ,OTL(CommOverCurrentConditionInProcess) ] ,XIO(UsingAgents) [OTL(CommOverCurrentConditionEventSuccess) ,OTU(CommOverCurrentConditionInProcess) ,OTE(CommuserNotified) ] ];
   // DCMicroGrid.Loads.Comm
   30: XIC(CommOverCurrentConditionInProcess)XIC(CommOverCurrentConditionEventSuccess)TON(CommOverCurrentConditionSuccessTimer,?,?);
   // DCMicroGrid.Loads.Comm
   31: XIC(CommOverCurrentConditionInProcess)XIC(CommOverCurrentConditionEventFail)TON(CommOverCurrentConditionFailTimer,?,?);
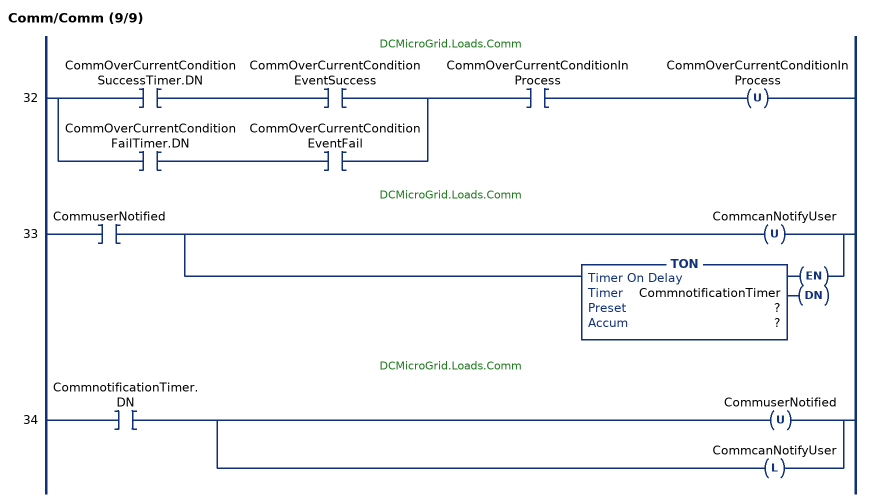
   // DCMicroGrid.Loads.Comm
   32: [XIC(CommOverCurrentConditionSuccessTimer.DN) XIC(CommOverCurrentConditionEventSuccess) ,XIC(CommOverCurrentConditionFailTimer.DN) XIC(CommOverCurrentConditionEventFail) ]XIC(CommOverCurrentConditionInProcess)OTU(CommOverCurrentConditionInProcess);
   // DCMicroGrid.Loads.Comm
   33: XIC(CommuserNotified)[OTU(CommcanNotifyUser) ,TON(CommnotificationTimer,?,?) ];
   // DCMicroGrid.Loads.Comm
   34: XIC(CommnotificationTimer.DN)[OTU(CommuserNotified) ,OTL(CommcanNotifyUser) ];
END_ROUTINE
END_PROGRAM
